TEXTLIST TextList_Servitudes
  0 = 'Groupe froid' | FR: 'Circulateur Chaud / Froid' | EN: 'Hot / Cold circulator'
  4 = '' | FR: "Tempéraure maximale de l'eau en sortie avant défaut" | EN: 'Maximum temperature for output water before fault'
  3 = '' | FR: "Tempéraure minimale de l'eau en sortie avant défaut" | EN: 'Minimum temperature for output water before fault'
  2 = '' | FR: "Débit maximal de l'eau en sortie avant défaut" | EN: 'Maximum flow for output water before fault'
  1 = '' | FR: "Débit minimal de l'eau en sortie avant défaut" | EN: 'Minimum flow for output water before fault'
  5 = '' | FR: "Tempéraure maximale de l'eau en sortie avant alarme" | EN: 'Maximum temperature for output water before warning'
   = ''
END_TEXTLIST

(* stored: Version 1.1.0.1, ProductVersion 3.1.4024.12
   TextList TextList_Servitudes: Id {f4e92ae0-b071-49b7-b6d9-7b2f6d419590} *)
